TYPE "PathTestSignal"
VERSION : 0.1
// Block: PathTestSignal
   STRUCT
      TestRequired : Bool;
      TestRunning : Bool;
      TestRunCmd : Bool;
   END_STRUCT;

END_TYPE
